{attribute 'qualified_only'}
VAR_GLOBAL
	// Case structure
	caseInput : INT := 0;
	
	// Variabelen
	ProductGedetecteerd1 : BOOL;	
	ProductGedetecteerd2 : BOOL;
	MotorStatus : BOOL;
	KlaarVoorVolgende : BOOL;

	// Timers
	Timer : TON;
	TimerOn : BOOL := FALSE;
END_VAR

(* stored: Version 1.1.0.1, ProductVersion 3.1.4024.12
   GVL GVL: Id {aa5d9f65-4fbf-4ab0-9237-d2df44e41fcb} *)
